# EPICS autosave request: 3-3/GalilSup/Db/galil_digital_out_bit.req
$(P)$(R)_CMD.VAL
$(P)$(R)_CMD.DESC
$(P)$(R)_STATUS.DESC
